// TIA Portal V15.1 export
// export: Created 2020-06-12T07:35:44.0693359Z, ExportSetting None, DisplayName Totally Integrated Automation Portal, DisplayVersion V15.1, DisplayName TIA Portal Openness, DisplayVersion V15.1, DisplayName STEP 7 Professional, DisplayVersion V15.1, DisplayName STEP 7 Safety, DisplayVersion V15.1, DisplayName WinCC Advanced, DisplayVersion V15.1
FUNCTION "PORT_HCC" : Void   // FC903, FBD
TITLE = High Current Return Clamp
{ S7_Optimized_Access := 'FALSE' }
// stored: AutoNumber false, SetENOAutomatically False
   VAR_TEMP
      tReady : Bool;
      _no_pos : Bool;
      _lock_melt : Bool;
      tClose1 : Bool;
      tOpen1 : Bool;
      tDeskActive : Bool;
      tClampsAreOpened : Bool;
      tClampsAreClosed : Bool;
      tClose2 : Bool;
      tOpen2 : Bool;
   END_VAR
BEGIN

REGION Network 1: common system fault
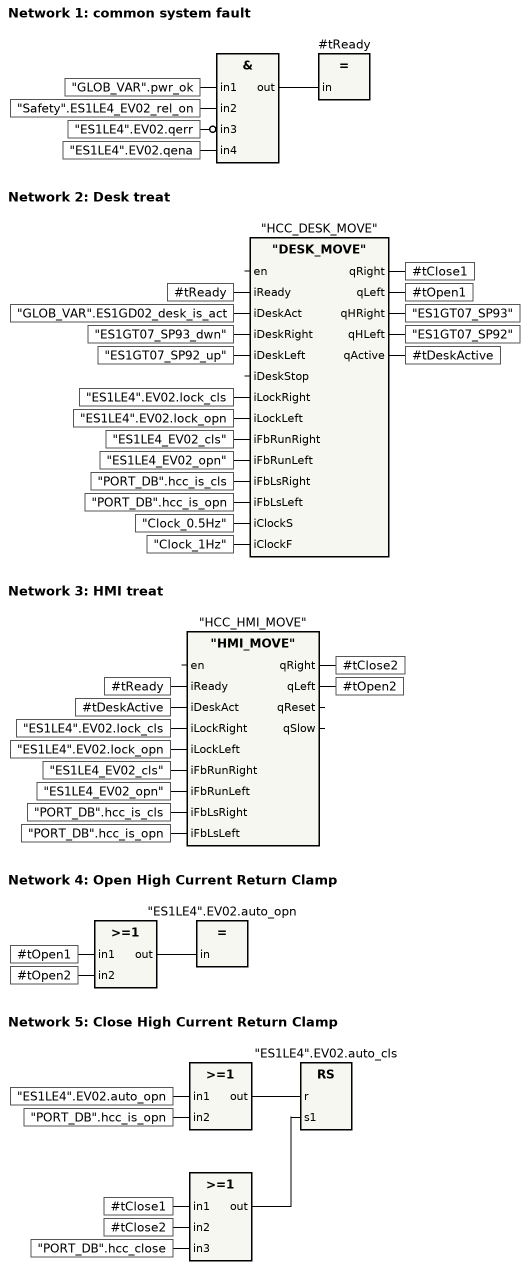
   #tReady := "GLOB_VAR".pwr_ok AND "Safety".ES1LE4_EV02_rel_on AND NOT "ES1LE4".EV02.qerr AND "ES1LE4".EV02.qena;
END_REGION

REGION Network 2: Desk treat
   "HCC_DESK_MOVE"(iReady := #tReady,   // "DESK_MOVE"
                   iDeskAct := "GLOB_VAR".ES1GD02_desk_is_act,
                   iDeskRight := "ES1GT07_SP93_dwn",
                   iDeskLeft := "ES1GT07_SP92_up",
                   iLockRight := "ES1LE4".EV02.lock_cls,
                   iLockLeft := "ES1LE4".EV02.lock_opn,
                   iFbRunRight := "ES1LE4_EV02_cls",
                   iFbRunLeft := "ES1LE4_EV02_opn",
                   iFbLsRight := "PORT_DB".hcc_is_cls,
                   iFbLsLeft := "PORT_DB".hcc_is_opn,
                   iClockS := "Clock_0.5Hz",
                   iClockF := "Clock_1Hz",
                   qRight => #tClose1,
                   qLeft => #tOpen1,
                   qHRight => "ES1GT07_SP93",
                   qHLeft => "ES1GT07_SP92",
                   qActive => #tDeskActive);
END_REGION

REGION Network 3: HMI treat
   "HCC_HMI_MOVE"(iReady := #tReady,   // "HMI_MOVE"
                  iDeskAct := #tDeskActive,
                  iLockRight := "ES1LE4".EV02.lock_cls,
                  iLockLeft := "ES1LE4".EV02.lock_opn,
                  iFbRunRight := "ES1LE4_EV02_cls",
                  iFbRunLeft := "ES1LE4_EV02_opn",
                  iFbLsRight := "PORT_DB".hcc_is_cls,
                  iFbLsLeft := "PORT_DB".hcc_is_opn,
                  qRight => #tClose2,
                  qLeft => #tOpen2);
END_REGION

REGION Network 4: Open High Current Return Clamp
   "ES1LE4".EV02.auto_opn := #tOpen1 OR #tOpen2;
END_REGION

REGION Network 5: Close High Current Return Clamp
   IF "ES1LE4".EV02.auto_opn OR "PORT_DB".hcc_is_opn THEN
       "ES1LE4".EV02.auto_cls := FALSE;   // RS flip-flop
   END_IF;
   IF #tClose1 OR #tClose2 OR "PORT_DB".hcc_close THEN "ES1LE4".EV02.auto_cls := TRUE; END_IF;
END_REGION

REGION Network 6: No definded Portal position
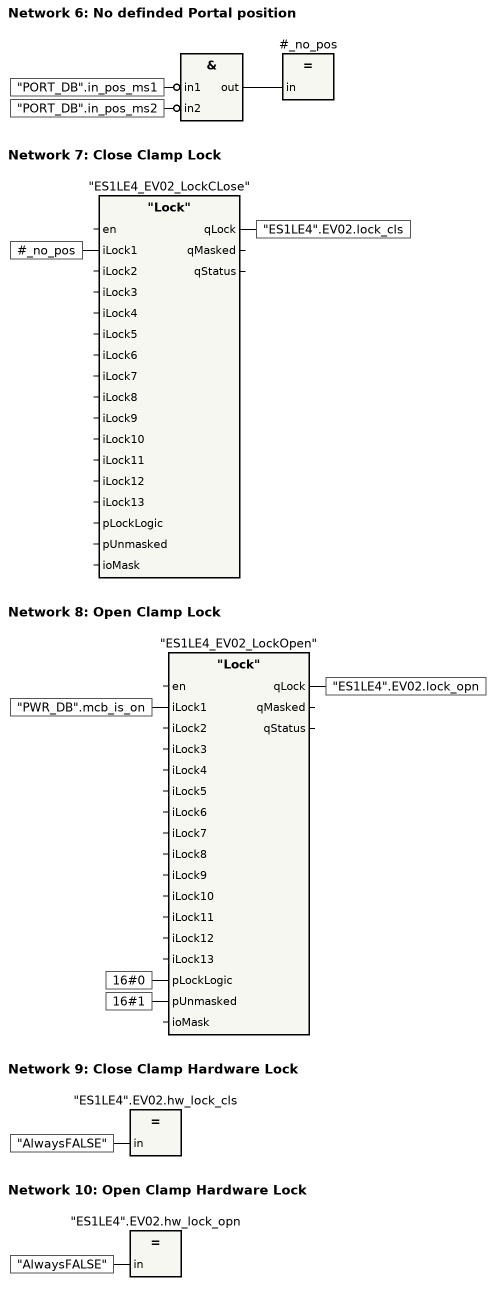
   #_no_pos := NOT "PORT_DB".in_pos_ms1 AND NOT "PORT_DB".in_pos_ms2;
END_REGION

REGION Network 7: Close Clamp Lock
   // "ES1LE4_PS02_pgmin_DI".qOUT
   "ES1LE4_EV02_LockCLose"(iLock1 := #_no_pos, qLock => "ES1LE4".EV02.lock_cls);   // "Lock"
END_REGION

REGION Network 8: Open Clamp Lock
   // VLS 08.05.2017: disable LOCK "Open
   "ES1LE4_EV02_LockOpen"(iLock1 := "PWR_DB".mcb_is_on,   // "Lock"
                          pLockLogic := 16#0,
                          pUnmasked := 16#1,
                          qLock => "ES1LE4".EV02.lock_opn);
END_REGION

REGION Network 9: Close Clamp Hardware Lock
   "ES1LE4".EV02.hw_lock_cls := "AlwaysFALSE";
END_REGION

REGION Network 10: Open Clamp Hardware Lock
   "ES1LE4".EV02.hw_lock_opn := "AlwaysFALSE";
END_REGION

REGION Network 11: Clamp is open
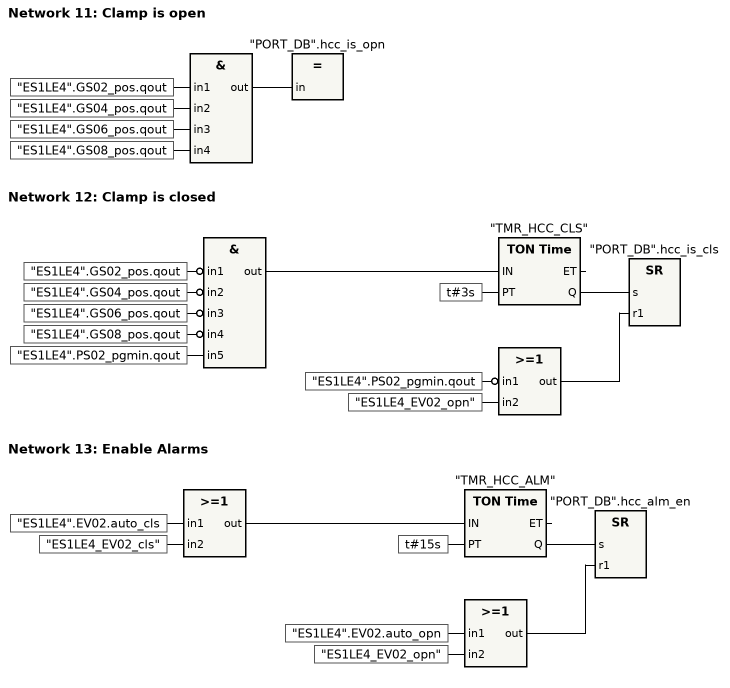
   "PORT_DB".hcc_is_opn := "ES1LE4".GS02_pos.qout AND "ES1LE4".GS04_pos.qout AND "ES1LE4".GS06_pos.qout AND "ES1LE4".GS08_pos.qout;
END_REGION

REGION Network 12: Clamp is closed
   "TMR_HCC_CLS".TON(IN := NOT "ES1LE4".GS02_pos.qout AND NOT "ES1LE4".GS04_pos.qout AND NOT "ES1LE4".GS06_pos.qout AND NOT "ES1LE4".GS08_pos.qout AND "ES1LE4".PS02_pgmin.qout,
                     PT := t#3s);
   IF "TMR_HCC_CLS".Q THEN
       "PORT_DB".hcc_is_cls := TRUE;   // SR flip-flop
   END_IF;
   IF NOT "ES1LE4".PS02_pgmin.qout OR "ES1LE4_EV02_opn" THEN "PORT_DB".hcc_is_cls := FALSE; END_IF;
END_REGION

REGION Network 13: Enable Alarms
   "TMR_HCC_ALM".TON(IN := "ES1LE4".EV02.auto_cls OR "ES1LE4_EV02_cls", PT := t#15s);
   IF "TMR_HCC_ALM".Q THEN
       "PORT_DB".hcc_alm_en := TRUE;   // SR flip-flop
   END_IF;
   IF "ES1LE4".EV02.auto_opn OR "ES1LE4_EV02_opn" THEN "PORT_DB".hcc_alm_en := FALSE; END_IF;
END_REGION
END_FUNCTION
